KUKA KRL data list: Zero_Position.dat

&ACCESS RV
&REL 1
DEFDAT Zero_Position PUBLIC
  DECL E6POS HOME={A1 0.0, A2 -90.0, A3 90.0, A4 0.0, A5 0.0, A6 0.0}
ENDDAT
